FUNCTION_BLOCK FB_Vereinzelung
VAR_INPUT
	//Steurervariablen
	bEnable : BOOL;
	bExecute : BOOL;
	
	//Hardwareeingänge
	bSensor1 : BOOL; //Flasche in der Kammer
	bSensor2 : BOOL; //Flasche im Rohr
	bSensor3 : BOOL; // Flasche auf Kopf
	bSensor4 : BOOL; // Flasche am Förderband
END_VAR
VAR_OUTPUT
	//Hardwareausgänge
	bGate1 : BOOL;
	bGate2 : BOOL;
	
	//Steuervariable
	eState : eBetriebszustand;
END_VAR
VAR
	nState : INT;
	fbTon : Ton;
END_VAR

fbTon(IN:= , PT:= T#1S, Q=> , ET=> );


CASE nState OF
	100: //Off / Nicht betriebsbereit
	eState := eBetriebszustand.Off;
	
	IF bSensor1 AND bEnable THEN
		nState := 21; //Ready
	ELSIF bEnable THEN
		nState := 0; //Init
	END_IF
	
	0: // Kammer ist leer
	eState := eBetriebszustand.Init;
	bGate1 := FALSE;
	bGate2 := FALSE;
	
	IF bSensor2 THEN
		nState := 1; //Oben öffnen
	END_IF
	
	1: //Oben öffnen
	eState := eBetriebszustand.Init;
	bGate1 := TRUE;
	bGate2 := FALSE;
	
	IF bSensor1 THEN
		nState := 2; // oben schließen
	END_IF
	
	2: //oben schließen
	eState := eBetriebszustand.Init;
	bGate1 := FALSE;
	bGate2 := FALSE;
	fbTon.IN := TRUE;
	
	IF fbTon.Q THEN
		nState := 21; //Ready
		fbTon.IN := FALSE;
		
	END_IF 
	
	21: //Ready
	eState := eBetriebszustand.Ready;
	bGate1 := FALSE;
	bGate2 := FALSE;
	fbTon.IN := TRUE;
	
	
	IF bExecute THEN
		nState:= 3;
	END_IF
	
	3:
	
	4:
	
END_CASE

END_FUNCTION_BLOCK

(* stored: Version 1.1.0.1, ProductVersion 3.1.4024.15
   POU FB_Vereinzelung: Id {127b2d98-2211-41c5-97cb-6f3fe87f5e4f}, SpecialFunc None *)
